// TIA Portal V20 export
TYPE "LWONIK_typeLaserInterlock"
// stored: Access Published
   STRUCT
      fromLaser_EstopOk : Bool;   // Laser Etop Ok Status
      fromLaser_EmissionOk : Bool;   // Laser Emission Ok Status
   END_STRUCT;
END_TYPE
